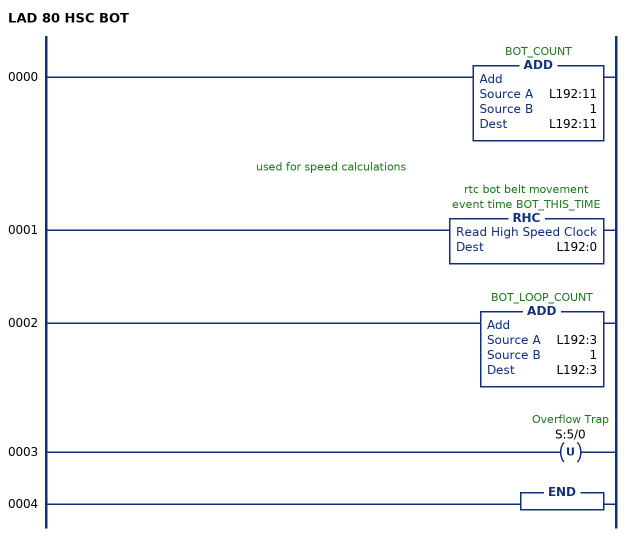
% Rung: 0 %
SOR ADD L192:11 1 L192:11 EOR
%   L192:11  BOT_COUNT %
% Rung: 1 %
% used for speed calculations %
SOR RHC L192:0 EOR
%   L192:0  BOT_THIS_TIME  "rtc bot belt movement event time" %
% Rung: 2 %
SOR ADD L192:3 1 L192:3 EOR
%   L192:3  BOT_LOOP_COUNT %
% Rung: 3 %
SOR OTU S:5/0 EOR
%   S:5/0  "Overflow Trap" %
% Rung: 4 %
SOR END EOR

LADDER 90 "HSC TOP"
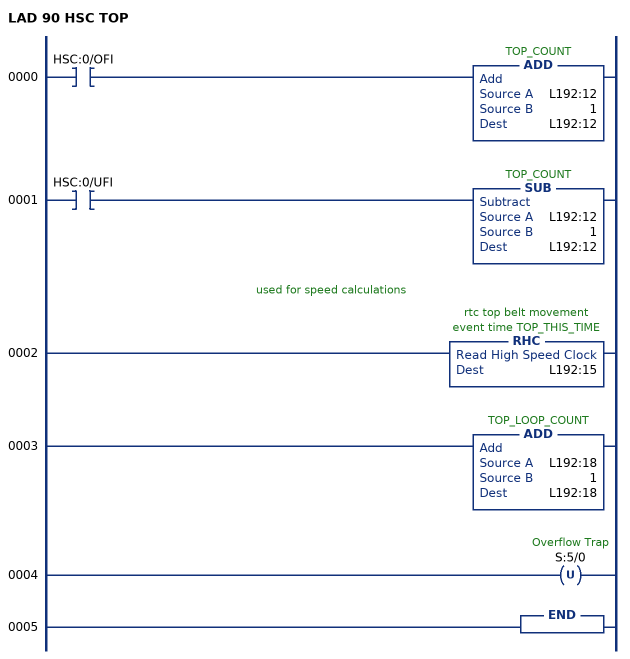
% Rung: 0 %
SOR XIC HSC:0/OFI ADD L192:12 1 L192:12 EOR
%   L192:12  TOP_COUNT %
% Rung: 1 %
SOR XIC HSC:0/UFI SUB L192:12 1 L192:12 EOR
%   L192:12  TOP_COUNT %
% Rung: 2 %
% used for speed calculations %
SOR RHC L192:15 EOR
%   L192:15  TOP_THIS_TIME  "rtc top belt movement event time" %
% Rung: 3 %
SOR ADD L192:18 1 L192:18 EOR
%   L192:18  TOP_LOOP_COUNT %
% Rung: 4 %
SOR OTU S:5/0 EOR
%   S:5/0  "Overflow Trap" %
% Rung: 5 %
SOR END EOR

LADDER 100 "1 MS STI"    % high speed %
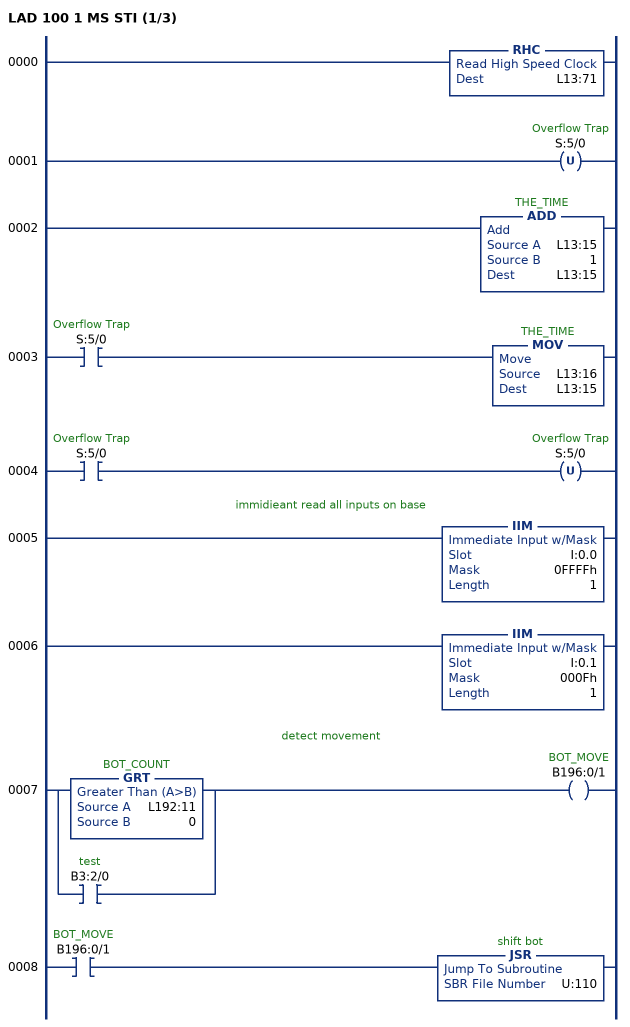
% Rung: 0 %
SOR RHC L13:71 EOR
% Rung: 1 %
SOR OTU S:5/0 EOR
%   S:5/0  "Overflow Trap" %
% Rung: 2 %
SOR ADD L13:15 1 L13:15 EOR
%   L13:15  THE_TIME %
% Rung: 3 %
SOR XIC S:5/0 MOV L13:16 L13:15 EOR
%   S:5/0  "Overflow Trap" %
%   L13:16  MIN_LONG %
%   L13:15  THE_TIME %
% Rung: 4 %
SOR XIC S:5/0 OTU S:5/0 EOR
%   S:5/0  "Overflow Trap" %
% Rung: 5 %
% immidieant read all inputs on base %
SOR IIM I:0.0 0FFFFh 1 EOR
% Rung: 6 %
SOR IIM I:0.1 000Fh 1 EOR
% Rung: 7 %
% detect movement %
SOR BST GRT L192:11 0 NXB XIC B3:2/0 BND OTE B196:0/1 EOR
%   L192:11  BOT_COUNT %
%   B3:2/0  "test" %
%   B196:0/1  BOT_MOVE %
% Rung: 8 %
SOR XIC B196:0/1 JSR U:110 EOR
%   B196:0/1  BOT_MOVE %
%   U:110  "shift bot" %

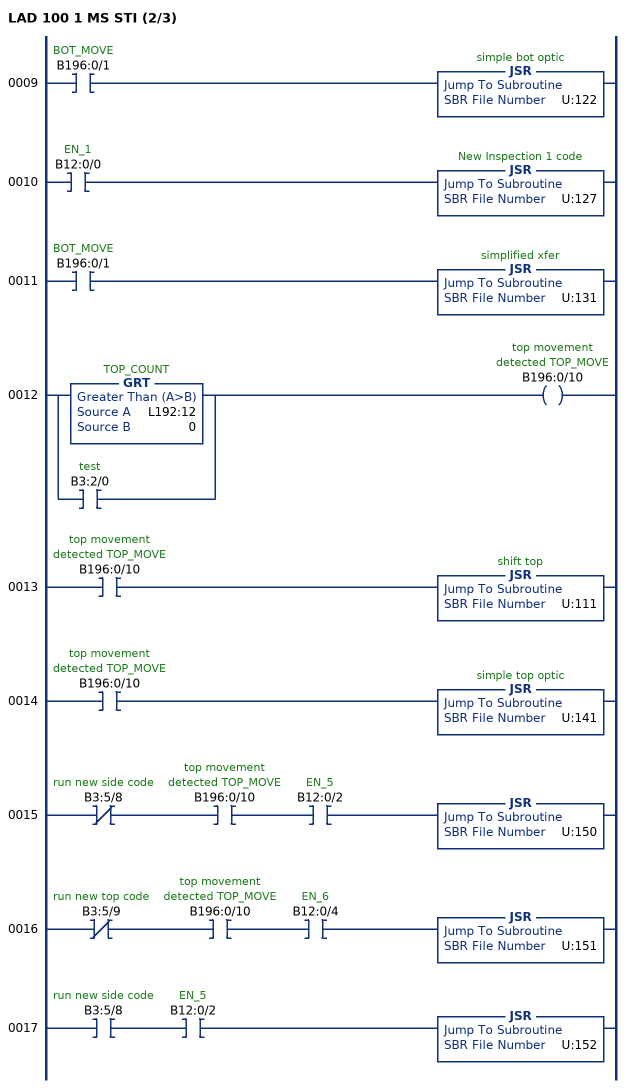
% Rung: 9 %
SOR XIC B196:0/1 JSR U:122 EOR
%   B196:0/1  BOT_MOVE %
%   U:122  "simple bot optic" %
% Rung: 10 %
SOR XIC B12:0/0 JSR U:127 EOR
%   B12:0/0  EN_1 %
%   U:127  "New Inspection 1 code" %
% Rung: 11 %
SOR XIC B196:0/1 JSR U:131 EOR
%   B196:0/1  BOT_MOVE %
%   U:131  "simplified xfer" %
% Rung: 12 %
SOR BST GRT L192:12 0 NXB XIC B3:2/0 BND OTE B196:0/10 EOR
%   L192:12  TOP_COUNT %
%   B3:2/0  "test" %
%   B196:0/10  TOP_MOVE  "top movement detected" %
% Rung: 13 %
SOR XIC B196:0/10 JSR U:111 EOR
%   B196:0/10  TOP_MOVE  "top movement detected" %
%   U:111  "shift top" %
% Rung: 14 %
SOR XIC B196:0/10 JSR U:141 EOR
%   B196:0/10  TOP_MOVE  "top movement detected" %
%   U:141  "simple top optic" %
% Rung: 15 %
SOR XIO B3:5/8 XIC B196:0/10 XIC B12:0/2 JSR U:150 EOR
%   B3:5/8  "run new side code" %
%   B196:0/10  TOP_MOVE  "top movement detected" %
%   B12:0/2  EN_5 %
% Rung: 16 %
SOR XIO B3:5/9 XIC B196:0/10 XIC B12:0/4 JSR U:151 EOR
%   B3:5/9  "run new top code" %
%   B196:0/10  TOP_MOVE  "top movement detected" %
%   B12:0/4  EN_6 %
% Rung: 17 %
SOR XIC B3:5/8 XIC B12:0/2 JSR U:152 EOR
%   B3:5/8  "run new side code" %
%   B12:0/2  EN_5 %

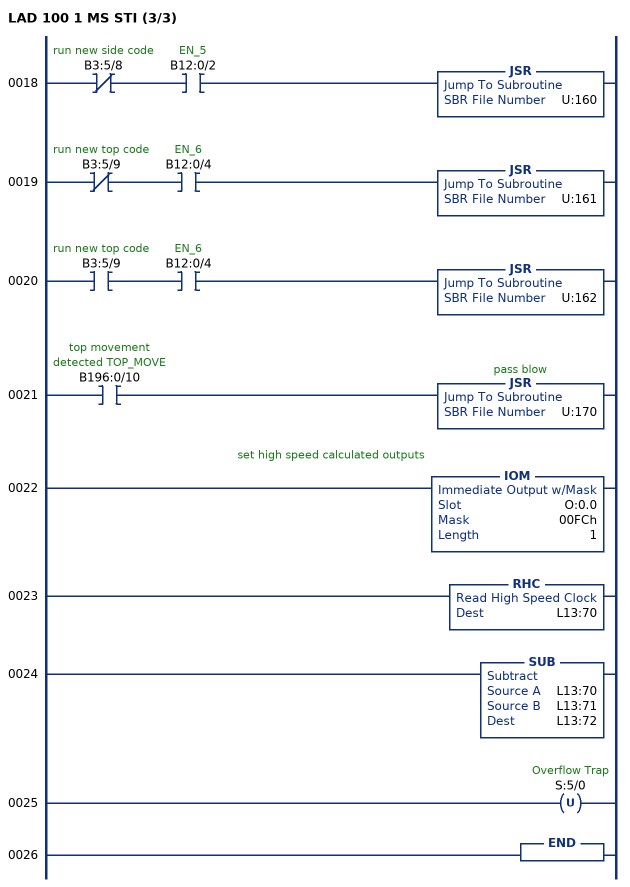
% Rung: 18 %
SOR XIO B3:5/8 XIC B12:0/2 JSR U:160 EOR
%   B3:5/8  "run new side code" %
%   B12:0/2  EN_5 %
% Rung: 19 %
SOR XIO B3:5/9 XIC B12:0/4 JSR U:161 EOR
%   B3:5/9  "run new top code" %
%   B12:0/4  EN_6 %
% Rung: 20 %
SOR XIC B3:5/9 XIC B12:0/4 JSR U:162 EOR
%   B3:5/9  "run new top code" %
%   B12:0/4  EN_6 %
% Rung: 21 %
SOR XIC B196:0/10 JSR U:170 EOR
%   B196:0/10  TOP_MOVE  "top movement detected" %
%   U:170  "pass blow" %
% Rung: 22 %
% set high speed calculated outputs %
SOR IOM O:0.0 00FCh 1 EOR
% Rung: 23 %
SOR RHC L13:70 EOR
% Rung: 24 %
SOR SUB L13:70 L13:71 L13:72 EOR
% Rung: 25 %
SOR OTU S:5/0 EOR
%   S:5/0  "Overflow Trap" %
% Rung: 26 %
SOR END EOR

LADDER 102 "SPEED BOT"    % high speed %
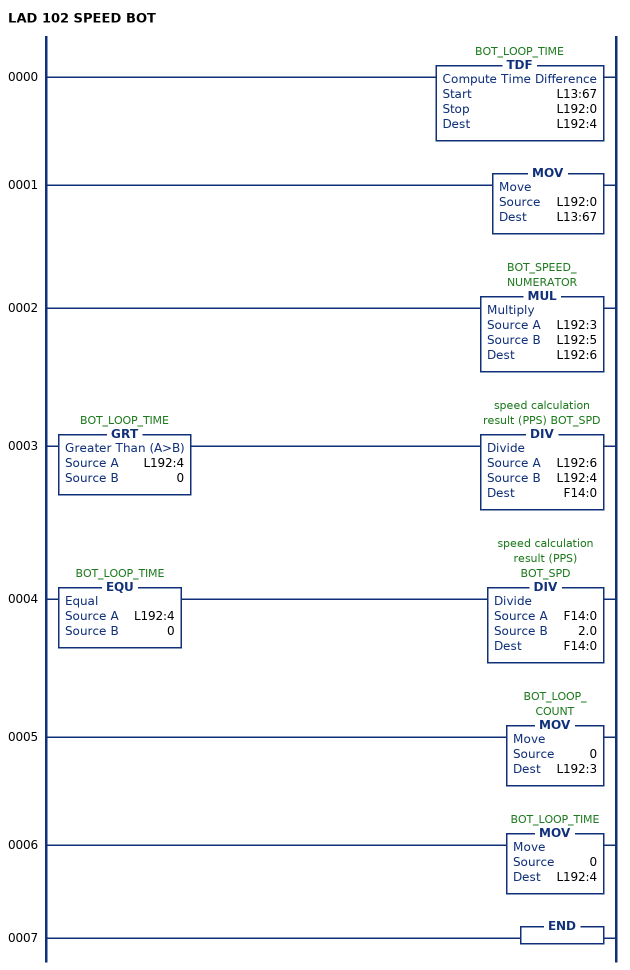
% Rung: 0 %
SOR TDF L13:67 L192:0 L192:4 EOR
%   L192:0  BOT_THIS_TIME  "rtc bot belt movement event time" %
%   L192:4  BOT_LOOP_TIME %
% Rung: 1 %
SOR MOV L192:0 L13:67 EOR
%   L192:0  BOT_THIS_TIME  "rtc bot belt movement event time" %
% Rung: 2 %
SOR MUL L192:3 L192:5 L192:6 EOR
%   L192:3  BOT_LOOP_COUNT %
%   L192:5  TKS_PER_SECOND %
%   L192:6  BOT_SPEED_NUMERATOR %
% Rung: 3 %
SOR GRT L192:4 0 DIV L192:6 L192:4 F14:0 EOR
%   L192:4  BOT_LOOP_TIME %
%   L192:6  BOT_SPEED_NUMERATOR %
%   F14:0  BOT_SPD  "speed calculation result (PPS)" %
% Rung: 4 %
SOR EQU L192:4 0 DIV F14:0 2.0 F14:0 EOR
%   L192:4  BOT_LOOP_TIME %
%   F14:0  BOT_SPD  "speed calculation result (PPS)" %
% Rung: 5 %
SOR MOV 0 L192:3 EOR
%   L192:3  BOT_LOOP_COUNT %
% Rung: 6 %
SOR MOV 0 L192:4 EOR
%   L192:4  BOT_LOOP_TIME %
% Rung: 7 %
SOR END EOR

LADDER 103 "SPEED TOP"    % high speed %
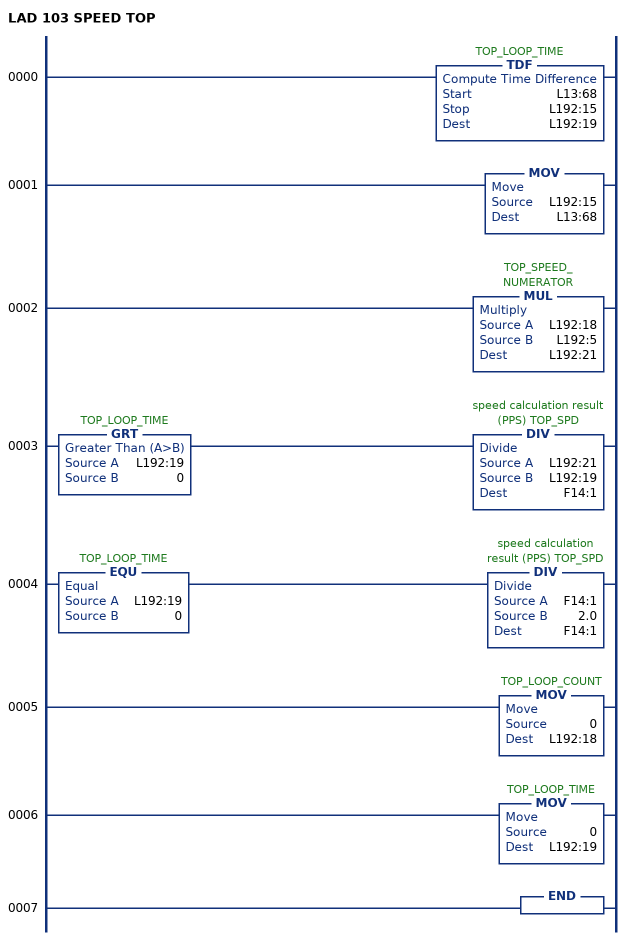
% Rung: 0 %
SOR TDF L13:68 L192:15 L192:19 EOR
%   L192:15  TOP_THIS_TIME  "rtc top belt movement event time" %
%   L192:19  TOP_LOOP_TIME %
% Rung: 1 %
SOR MOV L192:15 L13:68 EOR
%   L192:15  TOP_THIS_TIME  "rtc top belt movement event time" %
% Rung: 2 %
SOR MUL L192:18 L192:5 L192:21 EOR
%   L192:18  TOP_LOOP_COUNT %
%   L192:5  TKS_PER_SECOND %
%   L192:21  TOP_SPEED_NUMERATOR %
% Rung: 3 %
SOR GRT L192:19 0 DIV L192:21 L192:19 F14:1 EOR
%   L192:19  TOP_LOOP_TIME %
%   L192:21  TOP_SPEED_NUMERATOR %
%   F14:1  TOP_SPD  "speed calculation result (PPS)" %
% Rung: 4 %
SOR EQU L192:19 0 DIV F14:1 2.0 F14:1 EOR
%   L192:19  TOP_LOOP_TIME %
%   F14:1  TOP_SPD  "speed calculation result (PPS)" %
% Rung: 5 %
SOR MOV 0 L192:18 EOR
%   L192:18  TOP_LOOP_COUNT %
% Rung: 6 %
SOR MOV 0 L192:19 EOR
%   L192:19  TOP_LOOP_TIME %
% Rung: 7 %
SOR END EOR

LADDER 104 "P BOT"    % high speed %
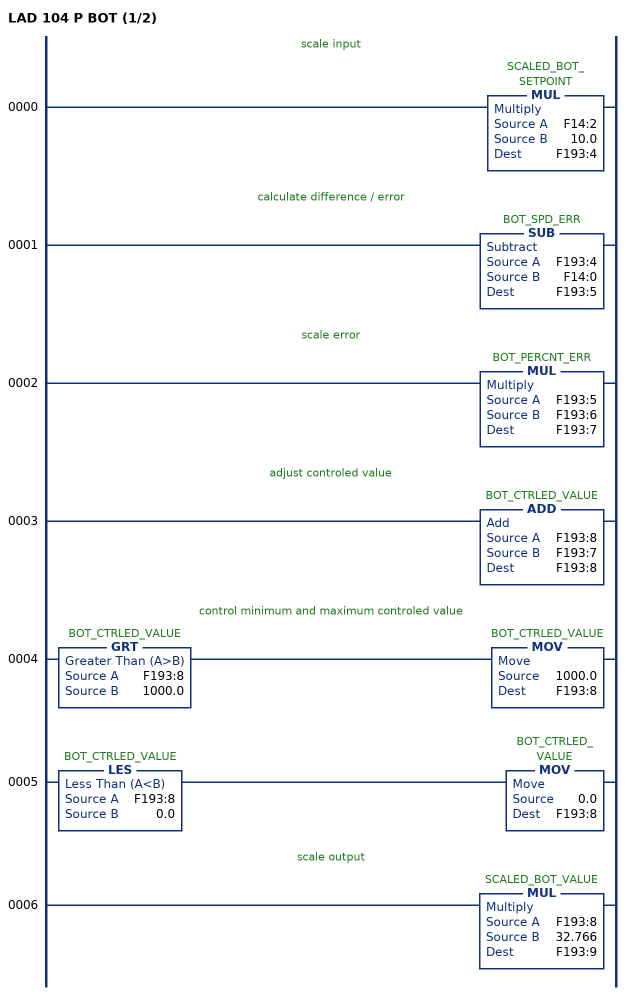
% Rung: 0 %
% scale input %
SOR MUL F14:2 10.0 F193:4 EOR
%   F14:2  BOT_SPD_SETPOINT %
%   F193:4  SCALED_BOT_SETPOINT %
% Rung: 1 %
% calculate difference / error %
SOR SUB F193:4 F14:0 F193:5 EOR
%   F193:4  SCALED_BOT_SETPOINT %
%   F14:0  BOT_SPD  "speed calculation result (PPS)" %
%   F193:5  BOT_SPD_ERR %
% Rung: 2 %
% scale error %
SOR MUL F193:5 F193:6 F193:7 EOR
%   F193:5  BOT_SPD_ERR %
%   F193:6  BOT_FDBK_RATIO %
%   F193:7  BOT_PERCNT_ERR %
% Rung: 3 %
% adjust controled value %
SOR ADD F193:8 F193:7 F193:8 EOR
%   F193:8  BOT_CTRLED_VALUE %
%   F193:7  BOT_PERCNT_ERR %
% Rung: 4 %
% control minimum and maximum controled value %
SOR GRT F193:8 1000.0 MOV 1000.0 F193:8 EOR
%   F193:8  BOT_CTRLED_VALUE %
% Rung: 5 %
SOR LES F193:8 0.0 MOV 0.0 F193:8 EOR
%   F193:8  BOT_CTRLED_VALUE %
% Rung: 6 %
% scale output %
SOR MUL F193:8 32.766 F193:9 EOR
%   F193:8  BOT_CTRLED_VALUE %
%   F193:9  SCALED_BOT_VALUE %

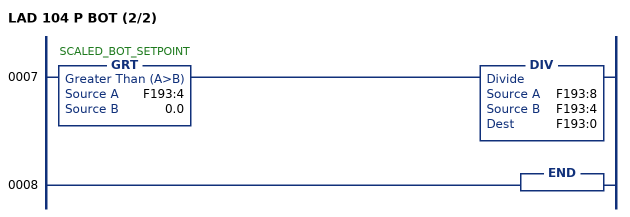
% Rung: 7 %
SOR GRT F193:4 0.0 DIV F193:8 F193:4 F193:0 EOR
%   F193:4  SCALED_BOT_SETPOINT %
%   F193:8  BOT_CTRLED_VALUE %
% Rung: 8 %
SOR END EOR

LADDER 105 "P TOP"    % high speed %
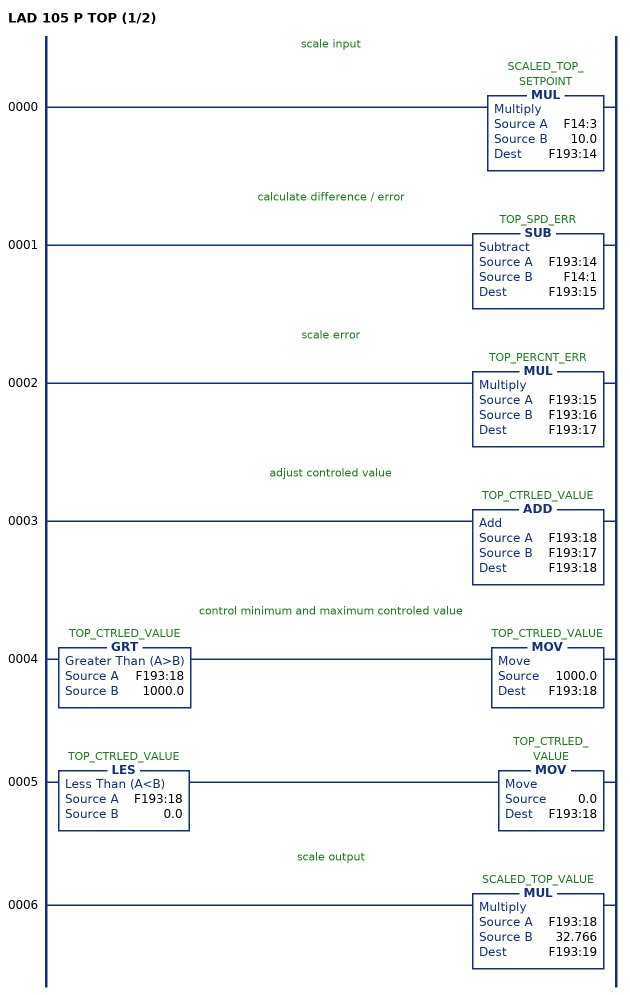
% Rung: 0 %
% scale input %
SOR MUL F14:3 10.0 F193:14 EOR
%   F14:3  TOP_SPD_SETPOINT %
%   F193:14  SCALED_TOP_SETPOINT %
% Rung: 1 %
% calculate difference / error %
SOR SUB F193:14 F14:1 F193:15 EOR
%   F193:14  SCALED_TOP_SETPOINT %
%   F14:1  TOP_SPD  "speed calculation result (PPS)" %
%   F193:15  TOP_SPD_ERR %
% Rung: 2 %
% scale error %
SOR MUL F193:15 F193:16 F193:17 EOR
%   F193:15  TOP_SPD_ERR %
%   F193:16  TOP_FDBK_RATIO %
%   F193:17  TOP_PERCNT_ERR %
% Rung: 3 %
% adjust controled value %
SOR ADD F193:18 F193:17 F193:18 EOR
%   F193:18  TOP_CTRLED_VALUE %
%   F193:17  TOP_PERCNT_ERR %
% Rung: 4 %
% control minimum and maximum controled value %
SOR GRT F193:18 1000.0 MOV 1000.0 F193:18 EOR
%   F193:18  TOP_CTRLED_VALUE %
% Rung: 5 %
SOR LES F193:18 0.0 MOV 0.0 F193:18 EOR
%   F193:18  TOP_CTRLED_VALUE %
% Rung: 6 %
% scale output %
SOR MUL F193:18 32.766 F193:19 EOR
%   F193:18  TOP_CTRLED_VALUE %
%   F193:19  SCALED_TOP_VALUE %

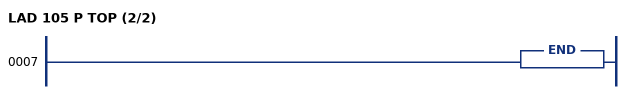
% Rung: 7 %
SOR END EOR

LADDER 110 "SHIFT BOT"
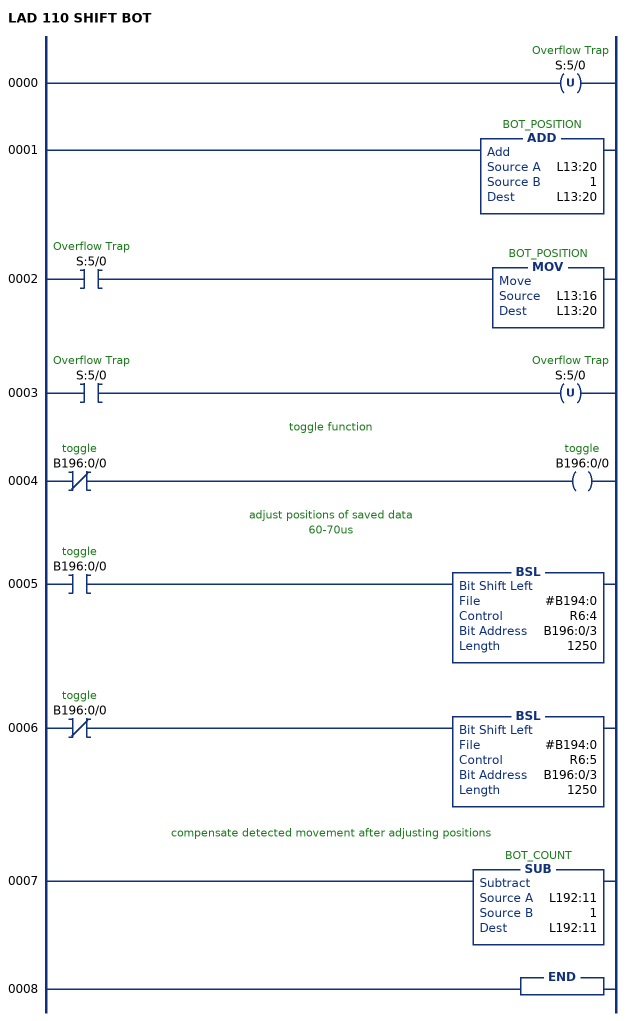
% Rung: 0 %
SOR OTU S:5/0 EOR
%   S:5/0  "Overflow Trap" %
% Rung: 1 %
SOR ADD L13:20 1 L13:20 EOR
%   L13:20  BOT_POSITION %
% Rung: 2 %
SOR XIC S:5/0 MOV L13:16 L13:20 EOR
%   S:5/0  "Overflow Trap" %
%   L13:16  MIN_LONG %
%   L13:20  BOT_POSITION %
% Rung: 3 %
SOR XIC S:5/0 OTU S:5/0 EOR
%   S:5/0  "Overflow Trap" %
% Rung: 4 %
% toggle function %
SOR XIO B196:0/0 OTE B196:0/0 EOR
%   B196:0/0  "toggle" %
% Rung: 5 %
% adjust positions of saved data
% 60-70us %
SOR XIC B196:0/0 BSL #B194:0 R6:4 B196:0/3 1250 EOR
%   B196:0/0  "toggle" %
%   B196:0/3  OFF %
% Rung: 6 %
SOR XIO B196:0/0 BSL #B194:0 R6:5 B196:0/3 1250 EOR
%   B196:0/0  "toggle" %
%   B196:0/3  OFF %
% Rung: 7 %
% compensate detected movement after adjusting positions %
SOR SUB L192:11 1 L192:11 EOR
%   L192:11  BOT_COUNT %
% Rung: 8 %
SOR END EOR

LADDER 111 "SHIFT TOP"
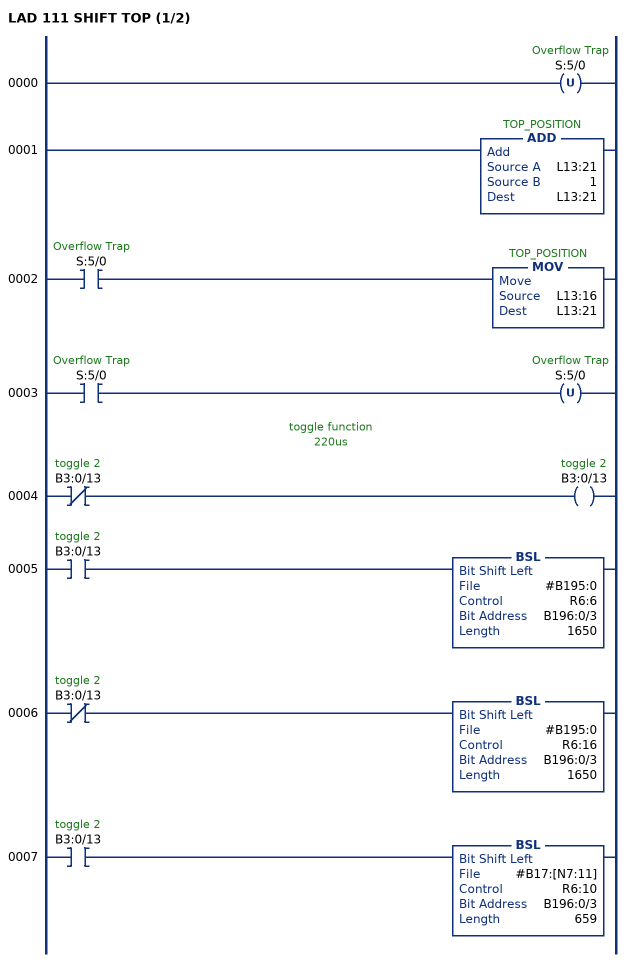
% Rung: 0 %
SOR OTU S:5/0 EOR
%   S:5/0  "Overflow Trap" %
% Rung: 1 %
SOR ADD L13:21 1 L13:21 EOR
%   L13:21  TOP_POSITION %
% Rung: 2 %
SOR XIC S:5/0 MOV L13:16 L13:21 EOR
%   S:5/0  "Overflow Trap" %
%   L13:16  MIN_LONG %
%   L13:21  TOP_POSITION %
% Rung: 3 %
SOR XIC S:5/0 OTU S:5/0 EOR
%   S:5/0  "Overflow Trap" %
% Rung: 4 %
% toggle function
% 220us %
SOR XIO B3:0/13 OTE B3:0/13 EOR
%   B3:0/13  "toggle 2" %
% Rung: 5 %
SOR XIC B3:0/13 BSL #B195:0 R6:6 B196:0/3 1650 EOR
%   B3:0/13  "toggle 2" %
%   R6:6  "from top load to top optic" %
%   B196:0/3  OFF %
% Rung: 6 %
SOR XIO B3:0/13 BSL #B195:0 R6:16 B196:0/3 1650 EOR
%   B3:0/13  "toggle 2" %
%   B196:0/3  OFF %
% Rung: 7 %
SOR XIC B3:0/13 BSL #B17:[N7:11] R6:10 B196:0/3 659 EOR
%   B3:0/13  "toggle 2" %
%   B196:0/3  OFF %

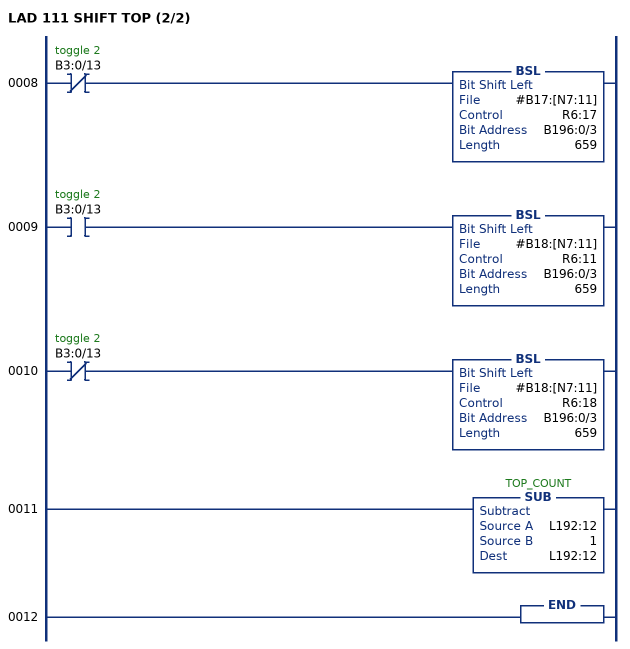
% Rung: 8 %
SOR XIO B3:0/13 BSL #B17:[N7:11] R6:17 B196:0/3 659 EOR
%   B3:0/13  "toggle 2" %
%   B196:0/3  OFF %
% Rung: 9 %
SOR XIC B3:0/13 BSL #B18:[N7:11] R6:11 B196:0/3 659 EOR
%   B3:0/13  "toggle 2" %
%   B196:0/3  OFF %
% Rung: 10 %
SOR XIO B3:0/13 BSL #B18:[N7:11] R6:18 B196:0/3 659 EOR
%   B3:0/13  "toggle 2" %
%   B196:0/3  OFF %
% Rung: 11 %
SOR SUB L192:12 1 L192:12 EOR
%   L192:12  TOP_COUNT %
% Rung: 12 %
SOR END EOR

LADDER 122 "OPTICBOT"
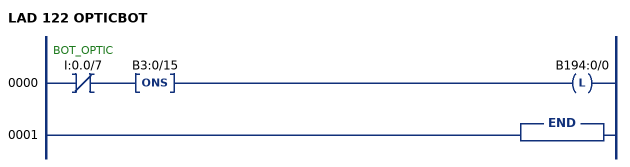
% Rung: 0 %
SOR XIO I:0.0/7 ONS B3:0/15 OTL B194:0/0 EOR
%   I:0.0/7  BOT_OPTIC %
% Rung: 1 %
SOR END EOR

LADDER 125 "INS 1 MOVE"
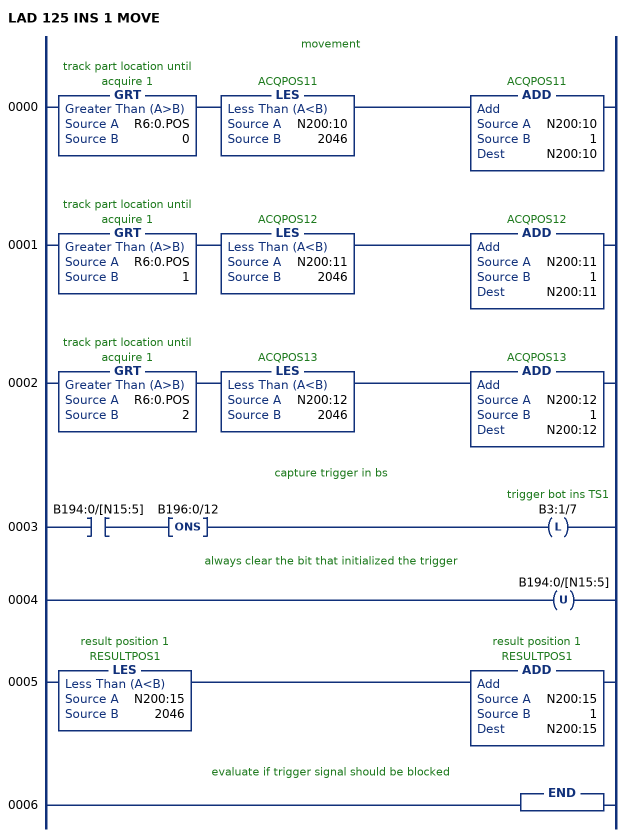
% Rung: 0 %
% movement %
SOR GRT R6:0.POS 0 LES N200:10 2046 ADD N200:10 1 N200:10 EOR
%   R6:0  "track part location until acquire 1" %
%   N200:10  ACQPOS11 %
% Rung: 1 %
SOR GRT R6:0.POS 1 LES N200:11 2046 ADD N200:11 1 N200:11 EOR
%   R6:0  "track part location until acquire 1" %
%   N200:11  ACQPOS12 %
% Rung: 2 %
SOR GRT R6:0.POS 2 LES N200:12 2046 ADD N200:12 1 N200:12 EOR
%   R6:0  "track part location until acquire 1" %
%   N200:12  ACQPOS13 %
% Rung: 3 %
% capture trigger in bs %
SOR XIC B194:0/[N15:5] ONS B196:0/12 OTL B3:1/7 EOR
%   N15:5  INS_1_TRIG_LOC %
%   B3:1/7  TS1  "trigger bot ins" %
% Rung: 4 %
% always clear the bit that initialized the trigger %
SOR OTU B194:0/[N15:5] EOR
%   N15:5  INS_1_TRIG_LOC %
% Rung: 5 %
SOR LES N200:15 2046 ADD N200:15 1 N200:15 EOR
%   N200:15  RESULTPOS1  "result position 1" %
% Rung: 6 %
% evaluate if trigger signal should be blocked %
SOR END EOR

LADDER 126 "INS 1TIME"
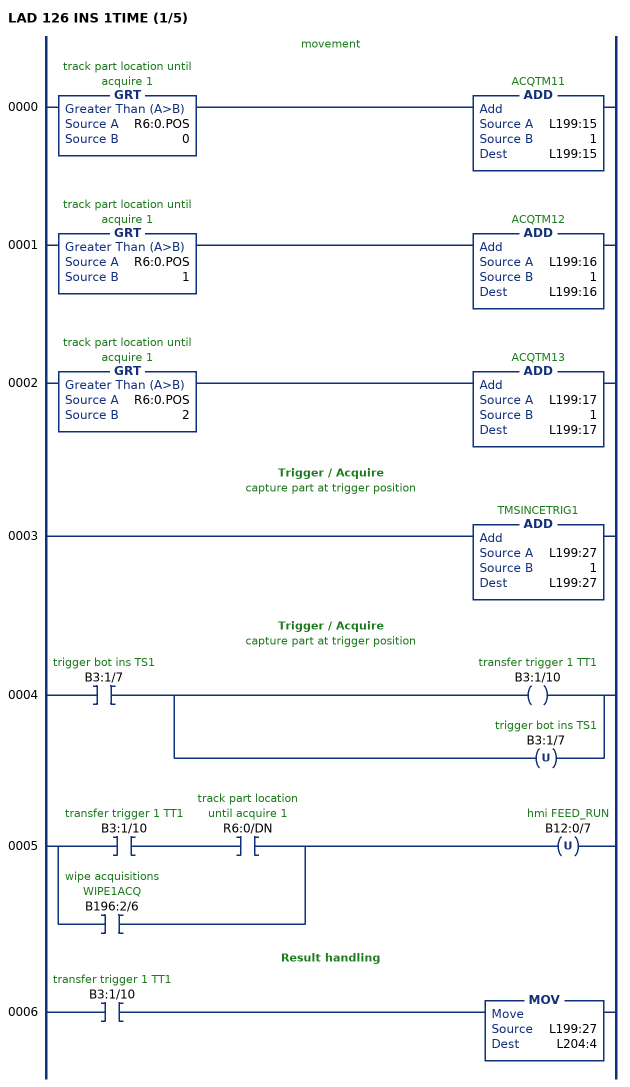
% Rung: 0 %
% movement %
SOR GRT R6:0.POS 0 ADD L199:15 1 L199:15 EOR
%   R6:0  "track part location until acquire 1" %
%   L199:15  ACQTM11 %
% Rung: 1 %
SOR GRT R6:0.POS 1 ADD L199:16 1 L199:16 EOR
%   R6:0  "track part location until acquire 1" %
%   L199:16  ACQTM12 %
% Rung: 2 %
SOR GRT R6:0.POS 2 ADD L199:17 1 L199:17 EOR
%   R6:0  "track part location until acquire 1" %
%   L199:17  ACQTM13 %
% Rung: 3 %
% TITLE: Trigger / Acquire %
% capture part at trigger position %
SOR ADD L199:27 1 L199:27 EOR
%   L199:27  TMSINCETRIG1 %
% Rung: 4 %
% TITLE: Trigger / Acquire %
% capture part at trigger position %
SOR XIC B3:1/7 BST OTE B3:1/10 NXB OTU B3:1/7 BND EOR
%   B3:1/7  TS1  "trigger bot ins" %
%   B3:1/10  TT1  "transfer trigger 1" %
% Rung: 5 %
SOR BST XIC B3:1/10 XIC R6:0/DN NXB XIC B196:2/6 BND OTU B12:0/7 EOR
%   B3:1/10  TT1  "transfer trigger 1" %
%   R6:0  "track part location until acquire 1" %
%   B196:2/6  WIPE1ACQ  "wipe acquisitions" %
%   B12:0/7  FEED_RUN  "hmi" %
% Rung: 6 %
% TITLE: Result handling %
SOR XIC B3:1/10 MOV L199:27 L204:4 EOR
%   B3:1/10  TT1  "transfer trigger 1" %
%   L199:27  TMSINCETRIG1 %

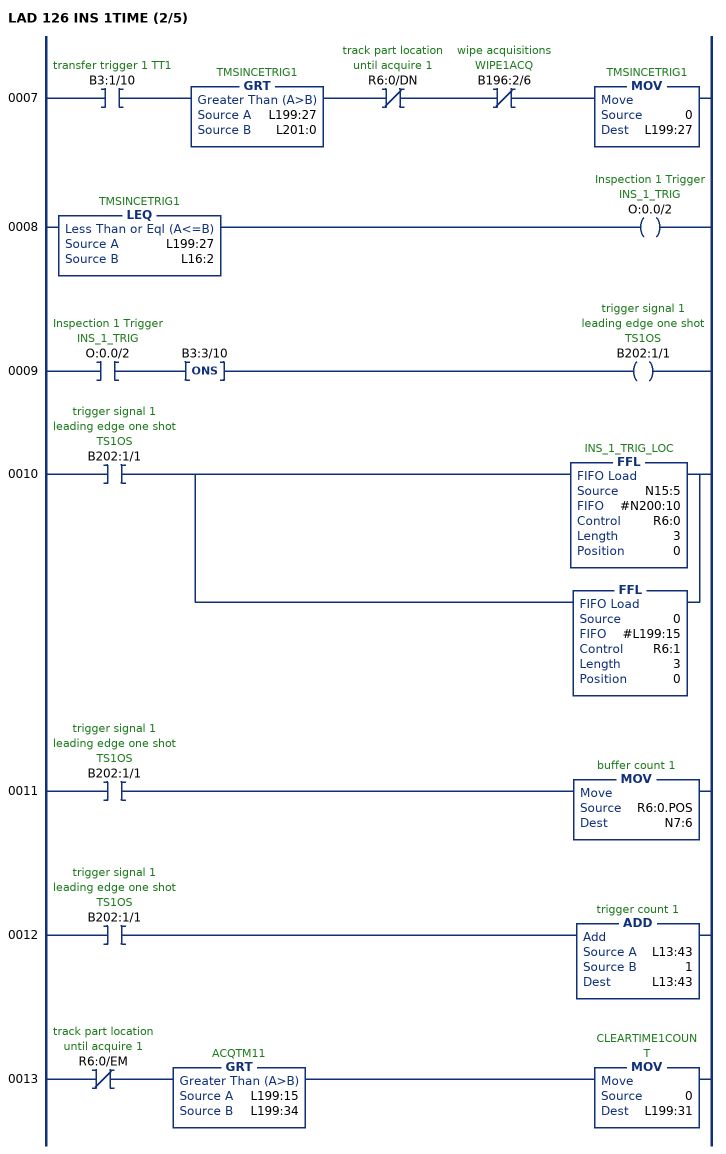
% Rung: 7 %
SOR XIC B3:1/10 GRT L199:27 L201:0 XIO R6:0/DN XIO B196:2/6 MOV 0 L199:27 EOR
%   B3:1/10  TT1  "transfer trigger 1" %
%   L199:27  TMSINCETRIG1 %
%   L201:0  CAM_1_MIN_CY %
%   R6:0  "track part location until acquire 1" %
%   B196:2/6  WIPE1ACQ  "wipe acquisitions" %
% Rung: 8 %
SOR LEQ L199:27 L16:2 OTE O:0.0/2 EOR
%   L199:27  TMSINCETRIG1 %
%   L16:2  CAM_1_TRIG_TIME %
%   O:0.0/2  INS_1_TRIG  "Inspection 1 Trigger" %
% Rung: 9 %
SOR XIC O:0.0/2 ONS B3:3/10 OTE B202:1/1 EOR
%   O:0.0/2  INS_1_TRIG  "Inspection 1 Trigger" %
%   B202:1/1  TS1OS  "trigger signal 1 leading edge one shot" %
% Rung: 10 %
SOR XIC B202:1/1 BST FFL N15:5 #N200:10 R6:0 3 0 NXB FFL 0 #L199:15 R6:1 3 0 BND EOR
%   B202:1/1  TS1OS  "trigger signal 1 leading edge one shot" %
%   N15:5  INS_1_TRIG_LOC %
%   N200:10  ACQPOS11 %
%   R6:0  "track part location until acquire 1" %
%   L199:15  ACQTM11 %
%   R6:1  "track acquire time 1" %
% Rung: 11 %
SOR XIC B202:1/1 MOV R6:0.POS N7:6 EOR
%   B202:1/1  TS1OS  "trigger signal 1 leading edge one shot" %
%   R6:0  "track part location until acquire 1" %
%   N7:6  "buffer count 1" %
% Rung: 12 %
SOR XIC B202:1/1 ADD L13:43 1 L13:43 EOR
%   B202:1/1  TS1OS  "trigger signal 1 leading edge one shot" %
%   L13:43  "trigger count 1" %
% Rung: 13 %
SOR XIO R6:0/EM GRT L199:15 L199:34 MOV 0 L199:31 EOR
%   R6:0  "track part location until acquire 1" %
%   L199:15  ACQTM11 %
%   L199:34  MAXACQTM1 %
%   L199:31  CLEARTIME1COUNT %

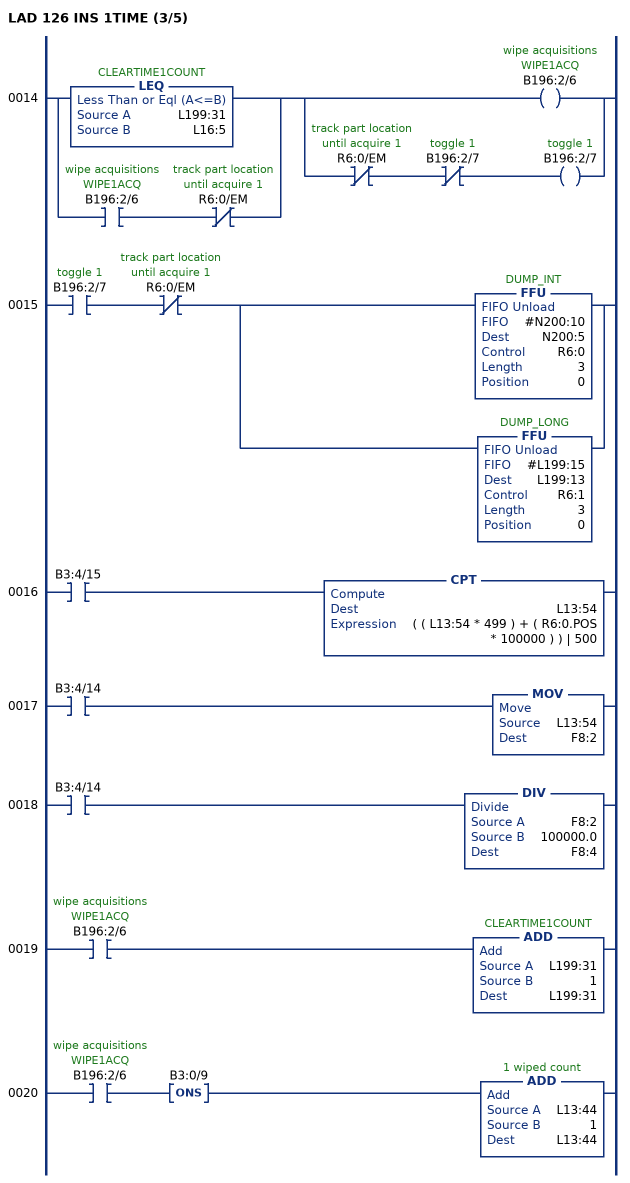
% Rung: 14 %
SOR BST LEQ L199:31 L16:5 NXB XIC B196:2/6 XIO R6:0/EM BND BST OTE B196:2/6 NXB XIO R6:0/EM XIO B196:2/7 OTE B196:2/7 BND EOR
%   L199:31  CLEARTIME1COUNT %
%   L16:5  CLEARTIME1  "time to clear tracking data" %
%   B196:2/6  WIPE1ACQ  "wipe acquisitions" %
%   R6:0  "track part location until acquire 1" %
%   B196:2/7  "toggle 1" %
% Rung: 15 %
SOR XIC B196:2/7 XIO R6:0/EM BST FFU #N200:10 N200:5 R6:0 3 0 NXB FFU #L199:15 L199:13 R6:1 3 0 BND EOR
%   B196:2/7  "toggle 1" %
%   R6:0  "track part location until acquire 1" %
%   N200:10  ACQPOS11 %
%   N200:5  DUMP_INT %
%   L199:15  ACQTM11 %
%   L199:13  DUMP_LONG %
%   R6:1  "track acquire time 1" %
% Rung: 16 %
SOR XIC B3:4/15 CPT L13:54 " ( ( L13:54 * 499 ) + ( R6:0.POS * 100000 ) ) | 500 " EOR
%   R6:0  "track part location until acquire 1" %
% Rung: 17 %
SOR XIC B3:4/14 MOV L13:54 F8:2 EOR
% Rung: 18 %
SOR XIC B3:4/14 DIV F8:2 100000.0 F8:4 EOR
% Rung: 19 %
SOR XIC B196:2/6 ADD L199:31 1 L199:31 EOR
%   B196:2/6  WIPE1ACQ  "wipe acquisitions" %
%   L199:31  CLEARTIME1COUNT %
% Rung: 20 %
SOR XIC B196:2/6 ONS B3:0/9 ADD L13:44 1 L13:44 EOR
%   B196:2/6  WIPE1ACQ  "wipe acquisitions" %
%   L13:44  "1 wiped count" %

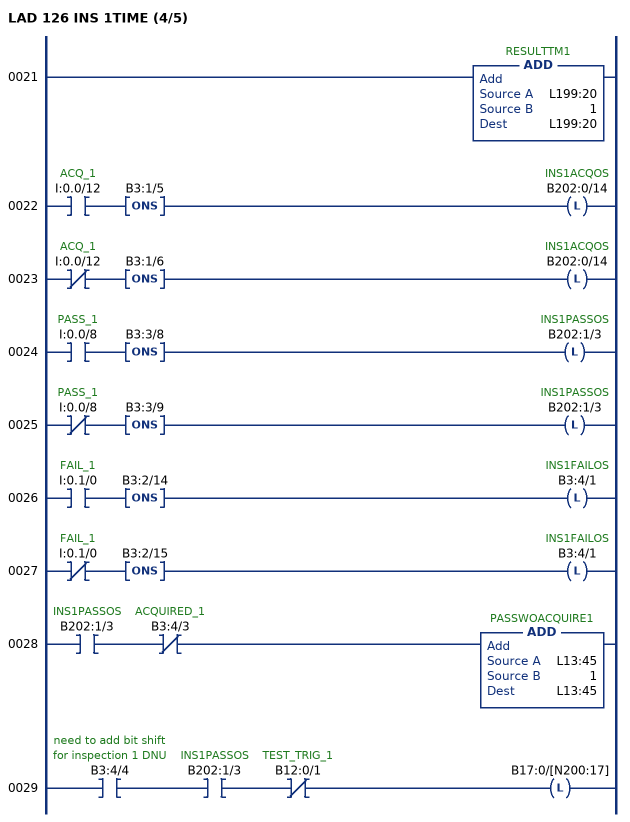
% Rung: 21 %
SOR ADD L199:20 1 L199:20 EOR
%   L199:20  RESULTTM1 %
% Rung: 22 %
SOR XIC I:0.0/12 ONS B3:1/5 OTL B202:0/14 EOR
%   I:0.0/12  ACQ_1 %
%   B202:0/14  INS1ACQOS %
% Rung: 23 %
SOR XIO I:0.0/12 ONS B3:1/6 OTL B202:0/14 EOR
%   I:0.0/12  ACQ_1 %
%   B202:0/14  INS1ACQOS %
% Rung: 24 %
SOR XIC I:0.0/8 ONS B3:3/8 OTL B202:1/3 EOR
%   I:0.0/8  PASS_1 %
%   B202:1/3  INS1PASSOS %
% Rung: 25 %
SOR XIO I:0.0/8 ONS B3:3/9 OTL B202:1/3 EOR
%   I:0.0/8  PASS_1 %
%   B202:1/3  INS1PASSOS %
% Rung: 26 %
SOR XIC I:0.1/0 ONS B3:2/14 OTL B3:4/1 EOR
%   I:0.1/0  FAIL_1 %
%   B3:4/1  INS1FAILOS %
% Rung: 27 %
SOR XIO I:0.1/0 ONS B3:2/15 OTL B3:4/1 EOR
%   I:0.1/0  FAIL_1 %
%   B3:4/1  INS1FAILOS %
% Rung: 28 %
SOR XIC B202:1/3 XIO B3:4/3 ADD L13:45 1 L13:45 EOR
%   B202:1/3  INS1PASSOS %
%   B3:4/3  ACQUIRED_1 %
%   L13:45  PASSWOACQUIRE1 %
% Rung: 29 %
SOR XIC B3:4/4 XIC B202:1/3 XIO B12:0/1 OTL B17:0/[N200:17] EOR
%   B3:4/4  DNU  "need to add bit shift for inspection 1" %
%   B202:1/3  INS1PASSOS %
%   B12:0/1  TEST_TRIG_1 %
%   N200:17  RESULTPOS5 %

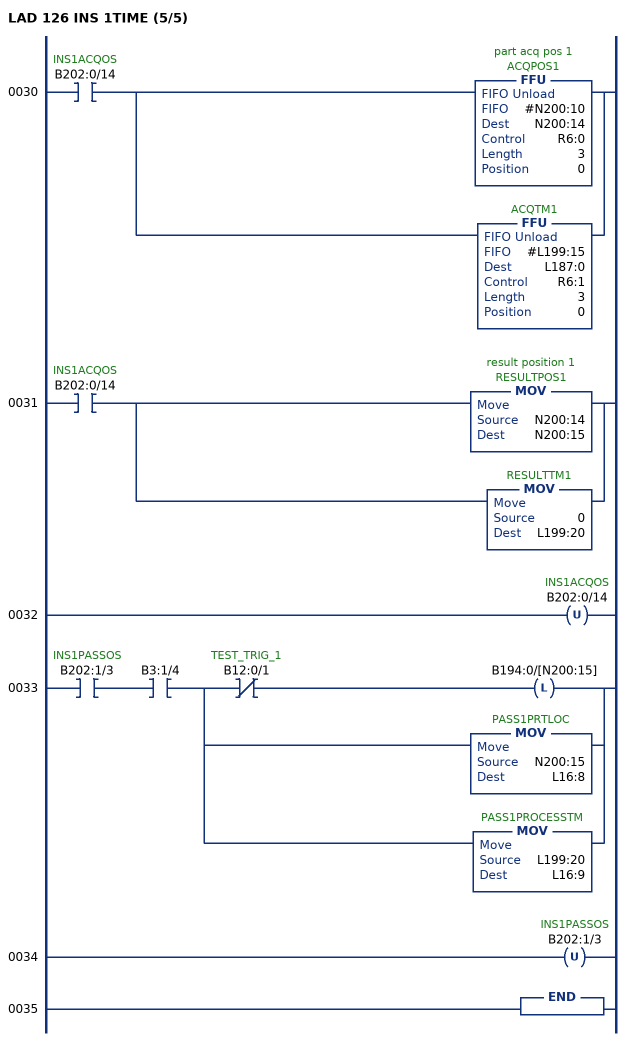
% Rung: 30 %
SOR XIC B202:0/14 BST FFU #N200:10 N200:14 R6:0 3 0 NXB FFU #L199:15 L187:0 R6:1 3 0 BND EOR
%   B202:0/14  INS1ACQOS %
%   N200:10  ACQPOS11 %
%   N200:14  ACQPOS1  "part acq pos 1" %
%   R6:0  "track part location until acquire 1" %
%   L199:15  ACQTM11 %
%   L187:0  ACQTM1 %
%   R6:1  "track acquire time 1" %
% Rung: 31 %
SOR XIC B202:0/14 BST MOV N200:14 N200:15 NXB MOV 0 L199:20 BND EOR
%   B202:0/14  INS1ACQOS %
%   N200:14  ACQPOS1  "part acq pos 1" %
%   N200:15  RESULTPOS1  "result position 1" %
%   L199:20  RESULTTM1 %
% Rung: 32 %
SOR OTU B202:0/14 EOR
%   B202:0/14  INS1ACQOS %
% Rung: 33 %
SOR XIC B202:1/3 XIC B3:1/4 BST XIO B12:0/1 OTL B194:0/[N200:15] NXB MOV N200:15 L16:8 NXB MOV L199:20 L16:9 BND EOR
%   B202:1/3  INS1PASSOS %
%   B12:0/1  TEST_TRIG_1 %
%   N200:15  RESULTPOS1  "result position 1" %
%   L16:8  PASS1PRTLOC %
%   L199:20  RESULTTM1 %
%   L16:9  PASS1PROCESSTM %
% Rung: 34 %
SOR OTU B202:1/3 EOR
%   B202:1/3  INS1PASSOS %
% Rung: 35 %
SOR END EOR

LADDER 127 "INS 1 NEW"
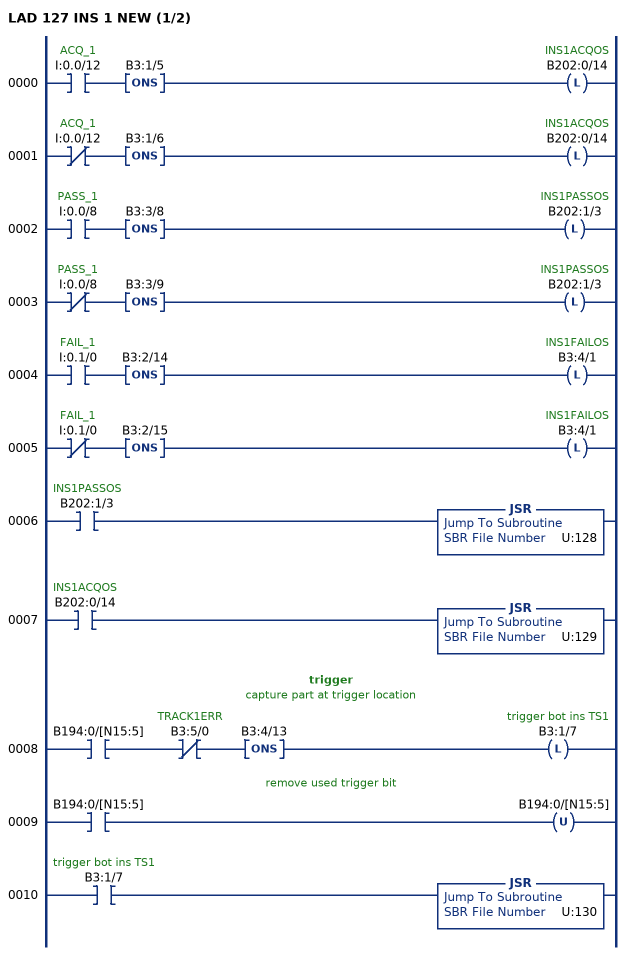
% Rung: 0 %
SOR XIC I:0.0/12 ONS B3:1/5 OTL B202:0/14 EOR
%   I:0.0/12  ACQ_1 %
%   B202:0/14  INS1ACQOS %
% Rung: 1 %
SOR XIO I:0.0/12 ONS B3:1/6 OTL B202:0/14 EOR
%   I:0.0/12  ACQ_1 %
%   B202:0/14  INS1ACQOS %
% Rung: 2 %
SOR XIC I:0.0/8 ONS B3:3/8 OTL B202:1/3 EOR
%   I:0.0/8  PASS_1 %
%   B202:1/3  INS1PASSOS %
% Rung: 3 %
SOR XIO I:0.0/8 ONS B3:3/9 OTL B202:1/3 EOR
%   I:0.0/8  PASS_1 %
%   B202:1/3  INS1PASSOS %
% Rung: 4 %
SOR XIC I:0.1/0 ONS B3:2/14 OTL B3:4/1 EOR
%   I:0.1/0  FAIL_1 %
%   B3:4/1  INS1FAILOS %
% Rung: 5 %
SOR XIO I:0.1/0 ONS B3:2/15 OTL B3:4/1 EOR
%   I:0.1/0  FAIL_1 %
%   B3:4/1  INS1FAILOS %
% Rung: 6 %
SOR XIC B202:1/3 JSR U:128 EOR
%   B202:1/3  INS1PASSOS %
% Rung: 7 %
SOR XIC B202:0/14 JSR U:129 EOR
%   B202:0/14  INS1ACQOS %
% Rung: 8 %
% TITLE: trigger %
% capture part at trigger location %
SOR XIC B194:0/[N15:5] XIO B3:5/0 ONS B3:4/13 OTL B3:1/7 EOR
%   N15:5  INS_1_TRIG_LOC %
%   B3:5/0  TRACK1ERR %
%   B3:1/7  TS1  "trigger bot ins" %
% Rung: 9 %
% remove used trigger bit %
SOR XIC B194:0/[N15:5] OTU B194:0/[N15:5] EOR
%   N15:5  INS_1_TRIG_LOC %
% Rung: 10 %
SOR XIC B3:1/7 JSR U:130 EOR
%   B3:1/7  TS1  "trigger bot ins" %

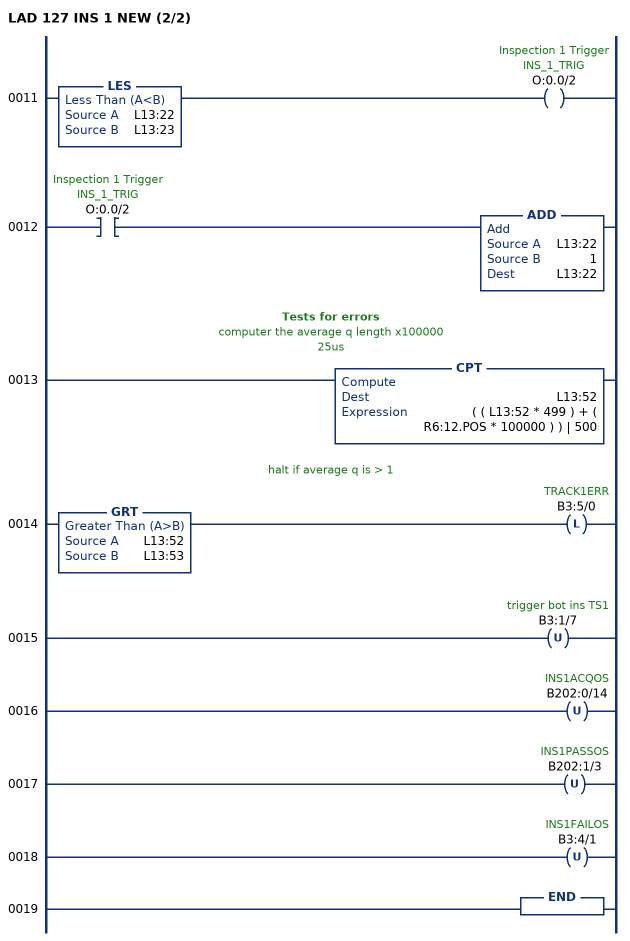
% Rung: 11 %
SOR LES L13:22 L13:23 OTE O:0.0/2 EOR
%   L13:23  "trigger on time" %
%   O:0.0/2  INS_1_TRIG  "Inspection 1 Trigger" %
% Rung: 12 %
SOR XIC O:0.0/2 ADD L13:22 1 L13:22 EOR
%   O:0.0/2  INS_1_TRIG  "Inspection 1 Trigger" %
% Rung: 13 %
% TITLE: Tests for errors %
% computer the average q length x100000
% 25us %
SOR CPT L13:52 " ( ( L13:52 * 499 ) + ( R6:12.POS * 100000 ) ) | 500 " EOR
% Rung: 14 %
% halt if average q is > 1 %
SOR GRT L13:52 L13:53 OTL B3:5/0 EOR
%   B3:5/0  TRACK1ERR %
% Rung: 15 %
SOR OTU B3:1/7 EOR
%   B3:1/7  TS1  "trigger bot ins" %
% Rung: 16 %
SOR OTU B202:0/14 EOR
%   B202:0/14  INS1ACQOS %
% Rung: 17 %
SOR OTU B202:1/3 EOR
%   B202:1/3  INS1PASSOS %
% Rung: 18 %
SOR OTU B3:4/1 EOR
%   B3:4/1  INS1FAILOS %
% Rung: 19 %
SOR END EOR

LADDER 128 "INS1PASS"
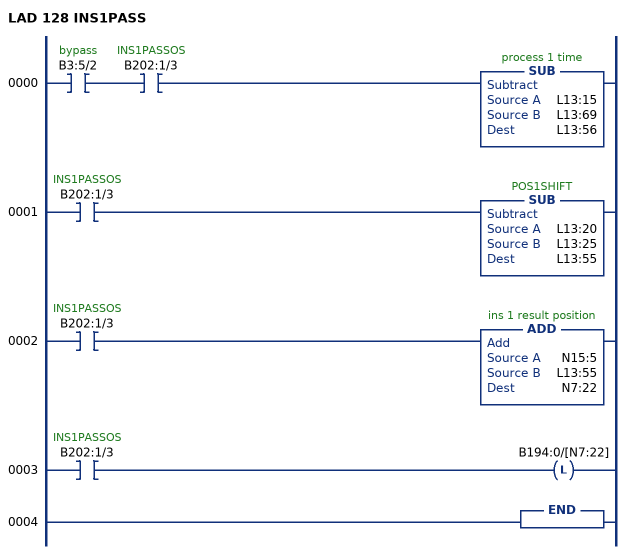
% Rung: 0 %
SOR XIC B3:5/2 XIC B202:1/3 SUB L13:15 L13:69 L13:56 EOR
%   B3:5/2  "bypass" %
%   B202:1/3  INS1PASSOS %
%   L13:15  THE_TIME %
%   L13:69  TIMEOFACQ1  "the time of the last acquire" %
%   L13:56  "process 1 time" %
% Rung: 1 %
SOR XIC B202:1/3 SUB L13:20 L13:25 L13:55 EOR
%   B202:1/3  INS1PASSOS %
%   L13:20  BOT_POSITION %
%   L13:25  POS1  "last acquisition position stamp" %
%   L13:55  POS1SHIFT %
% Rung: 2 %
SOR XIC B202:1/3 ADD N15:5 L13:55 N7:22 EOR
%   B202:1/3  INS1PASSOS %
%   N15:5  INS_1_TRIG_LOC %
%   L13:55  POS1SHIFT %
%   N7:22  "ins 1 result position" %
% Rung: 3 %
SOR XIC B202:1/3 OTL B194:0/[N7:22] EOR
%   B202:1/3  INS1PASSOS %
%   N7:22  "ins 1 result position" %
% Rung: 4 %
SOR END EOR

LADDER 129 "INS1ACQ"
